INTERFACE itfCamTable

METHOD Select		: itfCommand
VAR_INPUT
	Periodic		: BOOL;
	MasterAbsolute	: BOOL;
	SlaveAbsolute	: BOOL;
	CamTable		: MC_CAM_REF;
END_VAR
END_METHOD

END_INTERFACE

(* stored: Version 1.1.0.1, ProductVersion 3.1.4024.12
   Itf itfCamTable: Id {33c8a1dc-f227-43cf-8fb4-d9110092099b}
   Method Select: Id {8661899a-d268-40ac-b50a-0c4d39a150fe} *)
